ABB RAPID module: Module1.mod

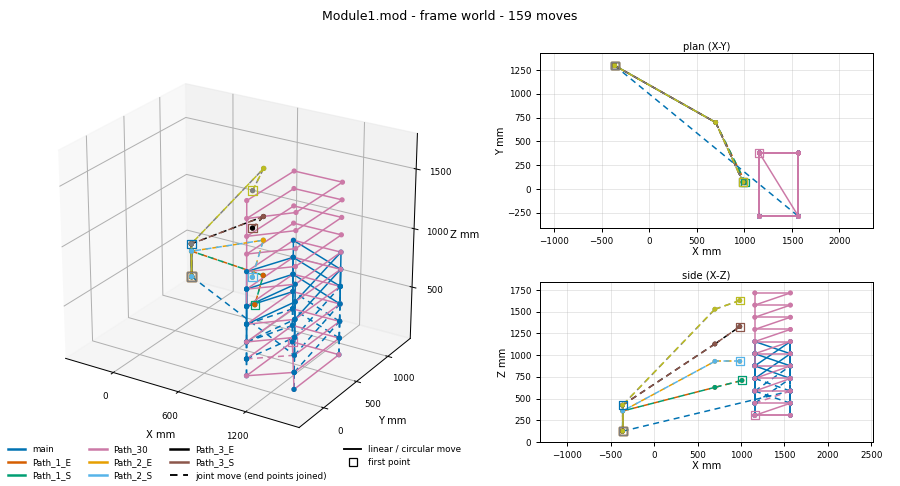
[picture p0: tool path of Module1.mod in frame world, 159 of 159 moves have a stored position in this frame; points joined in program order, loops and branches not executed]
MODULE Module1
        CONST robtarget Target_10:=[[-362.824,1298.255,124.558],[0,1,0,0],[0,0,0,0],[9E+09,9E+09,9E+09,9E+09,9E+09,9E+09]];
    CONST robtarget Target_20:=[[-361.331074857,1298.255015663,357.504486712],[0.000000006,0.937903782,0.346895511,-0.000000016],[1,0,-2,0],[9E+09,9E+09,9E+09,9E+09,9E+09,9E+09]];
    CONST robtarget Target_30:=[[699.999971128,699.99999496,629.43677315],[0.000000013,0.714564003,0.699570072,0.000000004],[0,-1,-2,0],[9E+09,9E+09,9E+09,9E+09,9E+09,9E+09]];
    CONST robtarget Target_50:=[[1570,-287,307],[0,0.707106781,0.707106781,0],[-1,0,0,0],[9E+09,9E+09,9E+09,9E+09,9E+09,9E+09]];
    CONST robtarget Target_40:=[[1012.141019914,68.859882763,709.132396194],[0.000000014,0.714564001,0.699570074,0.000000028],[0,0,-3,0],[9E+09,9E+09,9E+09,9E+09,9E+09,9E+09]];
    CONST robtarget Target_10_2:=[[-362.824,1298.255,424.558],[-0.000000012,0.998529603,-0.054209154,0.000000007],[1,0,-1,0],[9E+09,9E+09,9E+09,9E+09,9E+09,9E+09]];
    CONST robtarget Target_50_3:=[[1160,378,307],[0,0.707106781,0.707106781,0],[0,0,0,0],[9E+09,9E+09,9E+09,9E+09,9E+09,9E+09]];
    CONST robtarget Target_50_2:=[[1570,378,307],[0,0.707106781,0.707106781,0],[0,0,0,0],[9E+09,9E+09,9E+09,9E+09,9E+09,9E+09]];
    CONST robtarget Target_50_4:=[[1160,-287,307],[0,0.707106781,0.707106781,0],[-1,0,0,0],[9E+09,9E+09,9E+09,9E+09,9E+09,9E+09]];
    CONST robtarget Target_60:=[[1570,-287,447],[0,0.707106781,0.707106781,0],[0,0,0,0],[9E+09,9E+09,9E+09,9E+09,9E+09,9E+09]];
    CONST robtarget Target_60_2:=[[1570,378,447],[0,0.707106781,0.707106781,0],[0,0,1,0],[9E+09,9E+09,9E+09,9E+09,9E+09,9E+09]];
    CONST robtarget Target_60_3:=[[1160,378,447],[0,0.707106781,0.707106781,0],[0,0,1,0],[9E+09,9E+09,9E+09,9E+09,9E+09,9E+09]];
    CONST robtarget Target_60_4:=[[1160,-287,447],[0,0.707106781,0.707106781,0],[-1,0,0,0],[9E+09,9E+09,9E+09,9E+09,9E+09,9E+09]];
    CONST robtarget Target_120:=[[1570.000098335,-287.000000227,586.999987936],[-0.000000001,0.707106765,0.707106797,-0.000000001],[-1,-1,0,0],[9E+09,9E+09,9E+09,9E+09,9E+09,9E+09]];
    CONST robtarget Target_120_2:=[[1570,378,587],[0,0.707106781,0.707106781,0],[0,0,1,0],[9E+09,9E+09,9E+09,9E+09,9E+09,9E+09]];
    CONST robtarget Target_120_3:=[[1160,378,587],[0,0.707106781,0.707106781,0],[0,0,1,0],[9E+09,9E+09,9E+09,9E+09,9E+09,9E+09]];
    CONST robtarget Target_120_4:=[[1160,-287,587],[0,0.707106781,0.707106781,0],[-1,0,0,0],[9E+09,9E+09,9E+09,9E+09,9E+09,9E+09]];
    CONST robtarget Target_121:=[[1570,-287,732],[0,0.707106781,0.707106781,0],[-1,0,0,0],[9E+09,9E+09,9E+09,9E+09,9E+09,9E+09]];
    CONST robtarget Target_121_2:=[[1570,378,732],[0,0.707106781,0.707106781,0],[0,0,1,0],[9E+09,9E+09,9E+09,9E+09,9E+09,9E+09]];
    CONST robtarget Target_121_3:=[[1160,378,732],[0,0.707106781,0.707106781,0],[0,0,1,0],[9E+09,9E+09,9E+09,9E+09,9E+09,9E+09]];
    CONST robtarget Target_121_4:=[[1160,-287,732],[0,0.707106781,0.707106781,0],[-1,0,0,0],[9E+09,9E+09,9E+09,9E+09,9E+09,9E+09]];
    CONST robtarget Target_122:=[[1570,-287,877],[0,0.707106781,0.707106781,0],[-1,0,0,0],[9E+09,9E+09,9E+09,9E+09,9E+09,9E+09]];
    CONST robtarget Target_122_2:=[[1570,378,877],[0,0.707106781,0.707106781,0],[0,0,1,0],[9E+09,9E+09,9E+09,9E+09,9E+09,9E+09]];
    CONST robtarget Target_122_3:=[[1160,378,877],[0,0.707106781,0.707106781,0],[0,0,1,0],[9E+09,9E+09,9E+09,9E+09,9E+09,9E+09]];
    CONST robtarget Target_122_4:=[[1160,-287,877],[0,0.707106781,0.707106781,0],[-1,0,0,0],[9E+09,9E+09,9E+09,9E+09,9E+09,9E+09]];
    CONST robtarget Target_70_2:=[[699.999994937,700.000110159,929.436793547],[-0.000000013,0.714564003,0.699570072,0.000000004],[0,-1,-2,0],[9E+09,9E+09,9E+09,9E+09,9E+09,9E+09]];
    CONST robtarget Target_40_2:=[[987.25590411,72.978878039,929.436817205],[0.00000003,0.714563992,0.699570083,0.000000024],[0,-1,1,0],[9E+09,9E+09,9E+09,9E+09,9E+09,9E+09]];
    CONST robtarget Target_128_4:=[[1160,-287,1717],[0,0.707106781,0.707106781,0],[-1,2,-2,1],[9E+09,9E+09,9E+09,9E+09,9E+09,9E+09]];
    CONST robtarget Target_128_3:=[[1160,378,1717],[0,0.707106781,0.707106781,0],[0,0,1,0],[9E+09,9E+09,9E+09,9E+09,9E+09,9E+09]];
    CONST robtarget Target_128_2:=[[1570,378,1717],[0,0.707106781,0.707106781,0],[0,0,1,0],[9E+09,9E+09,9E+09,9E+09,9E+09,9E+09]];
    CONST robtarget Target_128:=[[1570,-287,1717],[0,0.707106781,0.707106781,0],[-1,0,0,0],[9E+09,9E+09,9E+09,9E+09,9E+09,9E+09]];
    CONST robtarget Target_127_4:=[[1160,-287,1577],[0,0.707106781,0.707106781,0],[-1,0,0,0],[9E+09,9E+09,9E+09,9E+09,9E+09,9E+09]];
    CONST robtarget Target_127_3:=[[1160,378,1577],[0,0.707106781,0.707106781,0],[0,0,1,0],[9E+09,9E+09,9E+09,9E+09,9E+09,9E+09]];
    CONST robtarget Target_127_2:=[[1570,378,1577],[0,0.707106781,0.707106781,0],[0,0,1,0],[9E+09,9E+09,9E+09,9E+09,9E+09,9E+09]];
    CONST robtarget Target_127:=[[1570,-287,1577],[0,0.707106781,0.707106781,0],[-1,0,0,0],[9E+09,9E+09,9E+09,9E+09,9E+09,9E+09]];
    CONST robtarget Target_126_4:=[[1160,-287,1437],[0,0.707106781,0.707106781,0],[-1,0,0,0],[9E+09,9E+09,9E+09,9E+09,9E+09,9E+09]];
    CONST robtarget Target_126_3:=[[1160,378,1437],[0,0.707106781,0.707106781,0],[0,0,1,0],[9E+09,9E+09,9E+09,9E+09,9E+09,9E+09]];
    CONST robtarget Target_126_2:=[[1570,378,1437],[0,0.707106781,0.707106781,0],[0,0,1,0],[9E+09,9E+09,9E+09,9E+09,9E+09,9E+09]];
    CONST robtarget Target_126:=[[1570,-287,1437],[0,0.707106781,0.707106781,0],[-1,0,0,0],[9E+09,9E+09,9E+09,9E+09,9E+09,9E+09]];
    CONST robtarget Target_125_4:=[[1160,-287,1297],[0,0.707106781,0.707106781,0],[-1,0,0,0],[9E+09,9E+09,9E+09,9E+09,9E+09,9E+09]];
    CONST robtarget Target_125_3:=[[1160,378,1297],[0,0.707106781,0.707106781,0],[0,0,1,0],[9E+09,9E+09,9E+09,9E+09,9E+09,9E+09]];
    CONST robtarget Target_125_2:=[[1570,378,1297],[0,0.707106781,0.707106781,0],[0,0,1,0],[9E+09,9E+09,9E+09,9E+09,9E+09,9E+09]];
    CONST robtarget Target_125:=[[1570,-287,1297],[0,0.707106781,0.707106781,0],[-1,0,0,0],[9E+09,9E+09,9E+09,9E+09,9E+09,9E+09]];
    CONST robtarget Target_124_4:=[[1160,-287,1157],[0,0.707106781,0.707106781,0],[-1,0,0,0],[9E+09,9E+09,9E+09,9E+09,9E+09,9E+09]];
    CONST robtarget Target_124_3:=[[1160,378,1157],[0,0.707106781,0.707106781,0],[0,0,1,0],[9E+09,9E+09,9E+09,9E+09,9E+09,9E+09]];
    CONST robtarget Target_124_2:=[[1570,378,1157],[0,0.707106781,0.707106781,0],[0,0,1,0],[9E+09,9E+09,9E+09,9E+09,9E+09,9E+09]];
    CONST robtarget Target_124:=[[1570,-287,1157],[0,0.707106781,0.707106781,0],[-1,0,0,0],[9E+09,9E+09,9E+09,9E+09,9E+09,9E+09]];
    CONST robtarget Target_123_4:=[[1160,-287,1017],[0,0.707106781,0.707106781,0],[-1,0,0,0],[9E+09,9E+09,9E+09,9E+09,9E+09,9E+09]];
    CONST robtarget Target_123_3:=[[1160,378,1017],[0,0.707106781,0.707106781,0],[0,0,1,0],[9E+09,9E+09,9E+09,9E+09,9E+09,9E+09]];
    CONST robtarget Target_123_2:=[[1570,378,1017],[0,0.707106781,0.707106781,0],[0,0,1,0],[9E+09,9E+09,9E+09,9E+09,9E+09,9E+09]];
    CONST robtarget Target_123:=[[1570,-287,1017],[0,0.707106781,0.707106781,0],[-1,0,0,0],[9E+09,9E+09,9E+09,9E+09,9E+09,9E+09]];
    CONST robtarget Target_30_2:=[[699.999992444,700.000011939,1129.436971585],[0.000000013,0.714563994,0.699570081,-0.000000007],[0,-1,-3,0],[9E+09,9E+09,9E+09,9E+09,9E+09,9E+09]];
    CONST robtarget Target_40_2_2:=[[987.255899553,72.978877702,1329.437041905],[0.00000002,0.714563994,0.699570081,0.000000013],[0,-1,1,0],[9E+09,9E+09,9E+09,9E+09,9E+09,9E+09]];
    CONST robtarget Target_10_4:=[[-362.824,1298.255,124.558],[0,1,0,0],[0,0,0,0],[9E+09,9E+09,9E+09,9E+09,9E+09,9E+09]];
    CONST robtarget Target_10_2_3:=[[-362.824,1298.255,424.558],[0,1,0,0],[1,0,-1,0],[9E+09,9E+09,9E+09,9E+09,9E+09,9E+09]];
    CONST robtarget Target_20_3:=[[123.294942114,850.000075451,439.015995707],[0.000000012,1,-0.000000212,0.000000031],[0,-1,-2,0],[9E+09,9E+09,9E+09,9E+09,9E+09,9E+09]];
    CONST robtarget Target_30_3:=[[699.999994518,700.000014013,1529.436978926],[0.000000013,0.714563998,0.699570077,0.000000012],[0,-1,-3,0],[9E+09,9E+09,9E+09,9E+09,9E+09,9E+09]];
    CONST robtarget Target_40_2_3:=[[987.255908383,72.978882952,1629.436986878],[-0.000000004,0.714563993,0.699570082,0.000000014],[0,0,1,0],[9E+09,9E+09,9E+09,9E+09,9E+09,9E+09]];
    CONST robtarget Target_20_2:=[[123.294942114,850.000075451,439.015995707],[0.000000013,0.714564003,0.699570072,0.000000004],[0,0,1,0],[9E+09,9E+09,9E+09,9E+09,9E+09,9E+09]];
    CONST robtarget Target_70:=[[700.00000486,700.000107801,929.436838226],[0.000000013,0.714563971,0.699570104,-0.000000014],[0,-1,-3,0],[9E+09,9E+09,9E+09,9E+09,9E+09,9E+09]];
!***********************************************************
    !
    ! Módulo:  Module1
    !
    ! Descripción:
    !   <Introduzca la descripción aquí>
    !
    ! Autor: deste
    !
    ! Versión: 1.0
    !
    !***********************************************************


    !***********************************************************
    !
    ! Procedimiento Main
    !
    !   Este es el punto de entrada de su programa
    !
    !***********************************************************
    PROC main()
        set Soltar;
        Reset Soltar;
        WaitDI Canasta_ok,1;
        MoveJ Target_10_2,v800,z100,Gripper\WObj:=Workobject_1;
        MoveL Target_10,v800,z100,Gripper\WObj:=Workobject_1;
        WaitUntil \InPos, Canasta_ok = 1;
        Set Agarrar;
        WaitDI Agarrado,1;
        Path_1_E;
        MoveJ Target_120,v800,z100,Gripper\WObj:=Workobject_1;
        MoveJ Target_60,v800,z10,Gripper\WObj:=Workobject_1;
        Reset Pallet;
        MoveJ Target_50,v800,z10,Gripper\WObj:=Workobject_1;
        WaitUntil \InPos, Canasta_ok = 0;
        Reset Agarrar;
        Set Soltar;
        Reset Soltar;
        MoveJ Target_60,v800,z100,Gripper\WObj:=Workobject_1;
        Path_1_S;
        !!! --------------------------- !!!
        WaitUntil \InPos, Canasta_ok = 1;
        Set Agarrar;
        WaitDI Agarrado,1;
        Path_1_E;
        MoveJ Target_120_2,v800,z100,Gripper\WObj:=Workobject_1;
        MoveJ Target_60_2,v800,z10,Gripper\WObj:=Workobject_1;
        Reset Pallet;
        MoveJ Target_50_2,v300,z10,Gripper\WObj:=Workobject_1;
        WaitUntil \InPos, Canasta_ok = 0;
        Reset Agarrar;
        Set Soltar;
        MoveJ Target_60_2,v800,z100,Gripper\WObj:=Workobject_1;
        Path_1_S;
        Reset Soltar;
        !!!-----------------------------!!!
        WaitUntil \InPos, Canasta_ok = 1;
        Set Agarrar;
        WaitDI Agarrado,1;
        Path_1_E;
        MoveJ Target_120_3,v800,z100,Gripper\WObj:=Workobject_1;
        MoveJ Target_60_3,v800,z10,Gripper\WObj:=Workobject_1;
        Reset Pallet;
        MoveJ Target_50_3,v300,z10,Gripper\WObj:=Workobject_1;
        WaitUntil \InPos, Canasta_ok = 0;
        Reset Agarrar;
        Set Soltar;
        MoveJ Target_60_3,v800,z100,Gripper\WObj:=Workobject_1;
        Path_1_S;
        Reset Soltar;
        !!!-----------------------------!!!
        WaitUntil \InPos, Canasta_ok = 1;
        Set Agarrar;
        WaitDI Agarrado,1;
        Path_1_E;
        MoveJ Target_120_4,v800,z100,Gripper\WObj:=Workobject_1;
        MoveJ Target_60_4,v800,z10,Gripper\WObj:=Workobject_1;
        Reset Pallet;
        MoveJ Target_50_4,v300,z10,Gripper\WObj:=Workobject_1;
        WaitUntil \InPos, Canasta_ok = 0;
        Reset Agarrar;
        Set Soltar;
        MoveJ Target_60_4,v800,z100,Gripper\WObj:=Workobject_1;
        Path_1_S;
        Reset Soltar;
        !!!-----------------------------!!! Segunda Bandeja
        WaitUntil \InPos, Canasta_ok = 1;
        Set Agarrar;
        WaitDI Agarrado,1;
        Path_1_E;
        MoveJ Target_121,v800,z100,Gripper\WObj:=Workobject_1;
        MoveJ Target_120,v800,z10,Gripper\WObj:=Workobject_1;
        Reset Pallet;
        MoveJ Target_60,v800,z10,Gripper\WObj:=Workobject_1;
        WaitUntil \InPos, Canasta_ok = 0;
        Reset Agarrar;
        Set Soltar;
        Reset Soltar;
        MoveJ Target_120,v800,z100,Gripper\WObj:=Workobject_1;
        Path_1_S;
        !!! --------------------------- !!!
        WaitUntil \InPos, Canasta_ok = 1;
        Set Agarrar;
        WaitDI Agarrado,1;
        Path_1_E;
        MoveJ Target_121_2,v800,z100,Gripper\WObj:=Workobject_1;
        MoveJ Target_120_2,v800,z10,Gripper\WObj:=Workobject_1;
        Reset Pallet;
        MoveJ Target_60_2,v300,z10,Gripper\WObj:=Workobject_1;
        WaitUntil \InPos, Canasta_ok = 0;
        Reset Agarrar;
        Set Soltar;
        MoveJ Target_120_2,v800,z100,Gripper\WObj:=Workobject_1;
        Path_1_S;
        Reset Soltar;
        !!!-----------------------------!!!
        WaitUntil \InPos, Canasta_ok = 1;
        Set Agarrar;
        WaitDI Agarrado,1;
        Path_1_E;
        MoveJ Target_121_3,v800,z100,Gripper\WObj:=Workobject_1;
        MoveJ Target_120_3,v800,z10,Gripper\WObj:=Workobject_1;
        Reset Pallet;
        MoveJ Target_60_3,v300,z10,Gripper\WObj:=Workobject_1;
        WaitUntil \InPos, Canasta_ok = 0;
        Reset Agarrar;
        Set Soltar;
        MoveJ Target_120_3,v800,z100,Gripper\WObj:=Workobject_1;
        Path_1_S;
        Reset Soltar;
        !!!-----------------------------!!!
        WaitUntil \InPos, Canasta_ok = 1;
        Set Agarrar;
        WaitDI Agarrado,1;
        Path_1_E;
        MoveJ Target_121_4,v800,z100,Gripper\WObj:=Workobject_1;
        MoveJ Target_120_4,v800,z10,Gripper\WObj:=Workobject_1;
        Reset Pallet;
        MoveJ Target_60_4,v300,z10,Gripper\WObj:=Workobject_1;
        WaitUntil \InPos, Canasta_ok = 0;
        Reset Agarrar;
        Set Soltar;
        MoveJ Target_120_4,v800,z100,Gripper\WObj:=Workobject_1;
        Path_1_S;
        Reset Soltar;
        !!!-----------------------------!!! Tercera Bandeja
        WaitUntil \InPos, Canasta_ok = 1;
        Set Agarrar;
        WaitDI Agarrado,1;
        Path_2_E;
        MoveJ Target_122,v800,z100,Gripper\WObj:=Workobject_1;
        MoveJ Target_121,v800,z10,Gripper\WObj:=Workobject_1;
        Reset Pallet;
        MoveL Target_120,v800,z10,Gripper\WObj:=Workobject_1;
        WaitUntil \InPos, Canasta_ok = 0;
        Reset Agarrar;
        Set Soltar;
        Reset Soltar;
        MoveJ Target_121,v800,z100,Gripper\WObj:=Workobject_1;
        Path_2_S;
        !!! --------------------------- !!!
        WaitUntil \InPos, Canasta_ok = 1;
        Set Agarrar;
        WaitDI Agarrado,1;
        Path_2_E;
        MoveJ Target_122_2,v800,z100,Gripper\WObj:=Workobject_1;
        MoveJ Target_121_2,v800,z10,Gripper\WObj:=Workobject_1;
        Reset Pallet;
        MoveJ Target_120_2,v300,z10,Gripper\WObj:=Workobject_1;
        WaitUntil \InPos, Canasta_ok = 0;
        Reset Agarrar;
        Set Soltar;
        MoveJ Target_121_2,v800,z100,Gripper\WObj:=Workobject_1;
        Path_2_S;
        Reset Soltar;
        !!!-----------------------------!!!
        WaitUntil \InPos, Canasta_ok = 1;
        Set Agarrar;
        WaitDI Agarrado,1;
        Path_2_E;
        MoveL Target_122_3,v800,z100,Gripper\WObj:=Workobject_1;
        MoveL Target_121_3,v800,z10,Gripper\WObj:=Workobject_1;
        Reset Pallet;
        MoveL Target_120_3,v300,z10,Gripper\WObj:=Workobject_1;
        WaitUntil \InPos, Canasta_ok = 0;
        Reset Agarrar;
        Set Soltar;
        MoveL Target_121_3,v800,z100,Gripper\WObj:=Workobject_1;
        Path_2_S;
        Reset Soltar;
        !!!-----------------------------!!!
        WaitUntil \InPos, Canasta_ok = 1;
        Set Agarrar;
        WaitDI Agarrado,1;
        Path_2_E;
        MoveL Target_122_4,v800,z100,Gripper\WObj:=Workobject_1;
        MoveL Target_121_4,v800,z10,Gripper\WObj:=Workobject_1;
        Reset Pallet;
        MoveL Target_120_4,v300,z10,Gripper\WObj:=Workobject_1;
        WaitUntil \InPos, Canasta_ok = 0;
        Reset Agarrar;
        Set Soltar;
        MoveL Target_121_4,v800,z100,Gripper\WObj:=Workobject_1;
        Path_2_S;
        Reset Soltar;
        !!!-----------------------------!!! Cuarta Bandeja
        WaitUntil \InPos, Canasta_ok = 1;
        Set Agarrar;
        WaitDI Agarrado,1;
        Path_2_E;
        MoveL Target_123,v800,z100,Gripper\WObj:=Workobject_1;
        MoveL Target_122,v800,z10,Gripper\WObj:=Workobject_1;
        Reset Pallet;
        MoveL Target_121,v800,z10,Gripper\WObj:=Workobject_1;
        WaitUntil \InPos, Canasta_ok = 0;
        Reset Agarrar;
        Set Soltar;
        Reset Soltar;
        MoveL Target_122,v800,z100,Gripper\WObj:=Workobject_1;
        Path_2_S;
        !!! --------------------------- !!!
        WaitUntil \InPos, Canasta_ok = 1;
        Set Agarrar;
        WaitDI Agarrado,1;
        Path_2_E;
        MoveL Target_123_2,v800,z100,Gripper\WObj:=Workobject_1;
        MoveL Target_122_2,v800,z10,Gripper\WObj:=Workobject_1;
        Reset Pallet;
        MoveL Target_121_2,v300,z10,Gripper\WObj:=Workobject_1;
        WaitUntil \InPos, Canasta_ok = 0;
        Reset Agarrar;
        Set Soltar;
        MoveL Target_122_2,v800,z100,Gripper\WObj:=Workobject_1;
        Path_2_S;
        Reset Soltar;
        !!!-----------------------------!!!
        WaitUntil \InPos, Canasta_ok = 1;
        Set Agarrar;
        WaitDI Agarrado,1;
        Path_2_E;
        MoveL Target_123_3,v800,z100,Gripper\WObj:=Workobject_1;
        MoveL Target_122_3,v800,z10,Gripper\WObj:=Workobject_1;
        Reset Pallet;
        MoveL Target_121_3,v300,z10,Gripper\WObj:=Workobject_1;
        WaitUntil \InPos, Canasta_ok = 0;
        Reset Agarrar;
        Set Soltar;
        MoveL Target_122_3,v800,z100,Gripper\WObj:=Workobject_1;
        Path_2_S;
        Reset Soltar;
        !!!-----------------------------!!!
        WaitUntil \InPos, Canasta_ok = 1;
        Set Agarrar;
        WaitDI Agarrado,1;
        Path_2_E;
        MoveL Target_123_4,v800,z100,Gripper\WObj:=Workobject_1;
        MoveL Target_122_4,v800,z10,Gripper\WObj:=Workobject_1;
        Reset Pallet;
        MoveL Target_121_4,v300,z10,Gripper\WObj:=Workobject_1;
        WaitUntil \InPos, Canasta_ok = 0;
        Reset Agarrar;
        Set Soltar;
        MoveL Target_122_4,v800,z100,Gripper\WObj:=Workobject_1;
        Path_2_S;
        Reset Soltar;
        !!!-----------------------------!!! Quinta Bandeja
        WaitUntil \InPos, Canasta_ok = 1;
        Set Agarrar;
        WaitDI Agarrado,1;
        Path_3_E;
        MoveL Target_124,v800,z100,Gripper\WObj:=Workobject_1;
        MoveL Target_123,v800,z10,Gripper\WObj:=Workobject_1;
        Reset Pallet;
        MoveL Target_122,v800,z10,Gripper\WObj:=Workobject_1;
        WaitUntil \InPos, Canasta_ok = 0;
        Reset Agarrar;
        Set Soltar;
        Reset Soltar;
        MoveL Target_123,v800,z100,Gripper\WObj:=Workobject_1;
        Path_3_S;
        !!! --------------------------- !!!
        WaitUntil \InPos, Canasta_ok = 1;
        Set Agarrar;
        WaitDI Agarrado,1;
        Path_3_E;
        MoveL Target_124_2,v800,z100,Gripper\WObj:=Workobject_1;
        MoveL Target_123_2,v800,z10,Gripper\WObj:=Workobject_1;
        Reset Pallet;
        MoveL Target_122_2,v300,z10,Gripper\WObj:=Workobject_1;
        WaitUntil \InPos, Canasta_ok = 0;
        Reset Agarrar;
        Set Soltar;
        MoveL Target_123_2,v800,z100,Gripper\WObj:=Workobject_1;
        Path_3_S;
        Reset Soltar;
        !!!-----------------------------!!!
        WaitUntil \InPos, Canasta_ok = 1;
        Set Agarrar;
        WaitDI Agarrado,1;
        Path_3_E;
        MoveL Target_124_3,v800,z100,Gripper\WObj:=Workobject_1;
        MoveL Target_123_3,v800,z10,Gripper\WObj:=Workobject_1;
        Reset Pallet;
        MoveL Target_122_3,v300,z10,Gripper\WObj:=Workobject_1;
        WaitUntil \InPos, Canasta_ok = 0;
        Reset Agarrar;
        Set Soltar;
        MoveL Target_123_3,v800,z100,Gripper\WObj:=Workobject_1;
        Path_3_S;
        Reset Soltar;
        !!!-----------------------------!!!
        WaitUntil \InPos, Canasta_ok = 1;
        Set Agarrar;
        WaitDI Agarrado,1;
        Path_3_E;
        MoveL Target_124_4,v800,z100,Gripper\WObj:=Workobject_1;
        MoveL Target_123_4,v800,z10,Gripper\WObj:=Workobject_1;
        Reset Pallet;
        MoveL Target_122_4,v300,z10,Gripper\WObj:=Workobject_1;
        WaitUntil \InPos, Canasta_ok = 0;
        Reset Agarrar;
        Set Soltar;
        MoveL Target_123_4,v800,z100,Gripper\WObj:=Workobject_1;
        Path_3_S;
        Reset Soltar;
    ENDPROC

    PROC Path_1_E()
        MoveL Target_10,v1000,z100,Gripper\WObj:=Workobject_1;
        MoveJ Target_20,v1000,z100,Gripper\WObj:=Workobject_1;
        MoveJ Target_30,v1000,z100,Gripper\WObj:=Workobject_1;
        MoveJ Target_40,v1000,z100,Gripper\WObj:=Workobject_1;
    ENDPROC
    PROC Path_1_S()
        MoveJ Target_40,v1000,z100,Gripper\WObj:=Workobject_1;
        MoveJ Target_30,v800,z100,Gripper\WObj:=Workobject_1;
        MoveJ Target_20,v1000,z100,Gripper\WObj:=Workobject_1;
        MoveJ Target_10,v600,z100,Gripper\WObj:=Workobject_1;
    ENDPROC
    PROC Path_30()
        MoveL Target_50_3,v1000,z100,Gripper\WObj:=Workobject_1;
        MoveL Target_50,v1000,z100,Gripper\WObj:=Workobject_1;
        MoveL Target_50_2,v1000,z100,Gripper\WObj:=Workobject_1;
        MoveL Target_50_3,v1000,z100,Gripper\WObj:=Workobject_1;
        MoveL Target_50_4,v1000,z100,Gripper\WObj:=Workobject_1;
        MoveL Target_60,v1000,z100,Gripper\WObj:=Workobject_1;
        MoveL Target_60_2,v1000,z100,Gripper\WObj:=Workobject_1;
        MoveL Target_60_3,v1000,z100,Gripper\WObj:=Workobject_1;
        MoveL Target_60_4,v1000,z100,Gripper\WObj:=Workobject_1;
        MoveJ Target_120,v1000,z100,Gripper\WObj:=Workobject_1;
        MoveL Target_120_2,v1000,z100,Gripper\WObj:=Workobject_1;
        MoveL Target_120_3,v1000,z100,Gripper\WObj:=Workobject_1;
        MoveL Target_120_4,v1000,z100,Gripper\WObj:=Workobject_1;
        MoveL Target_121,v1000,z100,Gripper\WObj:=Workobject_1;
        MoveL Target_121_2,v1000,z100,Gripper\WObj:=Workobject_1;
        MoveL Target_121_3,v1000,z100,Gripper\WObj:=Workobject_1;
        MoveL Target_121_4,v1000,z100,Gripper\WObj:=Workobject_1;
        MoveL Target_122,v1000,z100,Gripper\WObj:=Workobject_1;
        MoveL Target_122_2,v1000,z100,Gripper\WObj:=Workobject_1;
        MoveL Target_122_3,v1000,z100,Gripper\WObj:=Workobject_1;
        MoveL Target_122_4,v1000,z100,Gripper\WObj:=Workobject_1;
        MoveL Target_128_4,v1000,z100,Gripper\WObj:=Workobject_1;
        MoveL Target_128_3,v1000,z100,Gripper\WObj:=Workobject_1;
        MoveL Target_128_2,v1000,z100,Gripper\WObj:=Workobject_1;
        MoveL Target_128,v1000,z100,Gripper\WObj:=Workobject_1;
        MoveL Target_127_4,v1000,z100,Gripper\WObj:=Workobject_1;
        MoveL Target_127_3,v1000,z100,Gripper\WObj:=Workobject_1;
        MoveL Target_127_2,v1000,z100,Gripper\WObj:=Workobject_1;
        MoveL Target_127,v1000,z100,Gripper\WObj:=Workobject_1;
        MoveL Target_126_4,v1000,z100,Gripper\WObj:=Workobject_1;
        MoveL Target_126_3,v1000,z100,Gripper\WObj:=Workobject_1;
        MoveL Target_126_2,v1000,z100,Gripper\WObj:=Workobject_1;
        MoveL Target_126,v1000,z100,Gripper\WObj:=Workobject_1;
        MoveL Target_125_4,v1000,z100,Gripper\WObj:=Workobject_1;
        MoveL Target_125_3,v1000,z100,Gripper\WObj:=Workobject_1;
        MoveL Target_125_2,v1000,z100,Gripper\WObj:=Workobject_1;
        MoveL Target_125,v1000,z100,Gripper\WObj:=Workobject_1;
        MoveL Target_124_4,v1000,z100,Gripper\WObj:=Workobject_1;
        MoveL Target_124_3,v1000,z100,Gripper\WObj:=Workobject_1;
        MoveL Target_124_2,v1000,z100,Gripper\WObj:=Workobject_1;
        MoveL Target_124,v1000,z100,Gripper\WObj:=Workobject_1;
        MoveL Target_123_4,v1000,z100,Gripper\WObj:=Workobject_1;
        MoveL Target_123_3,v1000,z100,Gripper\WObj:=Workobject_1;
        MoveL Target_123_2,v1000,z100,Gripper\WObj:=Workobject_1;
        MoveL Target_123,v1000,z100,Gripper\WObj:=Workobject_1;
    ENDPROC
    PROC Path_2_E()
        MoveL Target_10,v1000,z100,Gripper\WObj:=Workobject_1;
        MoveJ Target_20,v1000,z100,Gripper\WObj:=Workobject_1;
        MoveJ Target_70,v1000,z100,Gripper\WObj:=Workobject_1;
        MoveJ Target_40_2,v1000,z100,Gripper\WObj:=Workobject_1;
    ENDPROC
    PROC Path_2_S()
        MoveL Target_40_2,v1000,z100,Gripper\WObj:=Workobject_1;
        MoveJ Target_70,v1000,z100,Gripper\WObj:=Workobject_1;
        MoveJ Target_20,v1000,z100,Gripper\WObj:=Workobject_1;
        MoveJ Target_10,v1000,z100,Gripper\WObj:=Workobject_1;
    ENDPROC
    PROC Path_3_E()
        MoveL Target_10,v1000,z100,Gripper\WObj:=Workobject_1;
        MoveL Target_10_2,v1000,z100,Gripper\WObj:=Workobject_1;
        MoveJ Target_30_2,v1000,z100,Gripper\WObj:=Workobject_1;
        MoveJ Target_40_2_2,v1000,z100,Gripper\WObj:=Workobject_1;
    ENDPROC
    PROC Path_3_S()
        MoveL Target_40_2_2,v1000,z100,Gripper\WObj:=Workobject_1;
        MoveJ Target_30_2,v1000,z100,Gripper\WObj:=Workobject_1;
        MoveJ Target_10_2,v1000,z100,Gripper\WObj:=Workobject_1;
        MoveL Target_10,v1000,z100,Gripper\WObj:=Workobject_1;
    ENDPROC
    PROC Path_4_E()
        MoveL Target_10_4,v1000,z100,Gripper\WObj:=Workobject_1;
        MoveL Target_10_2,v1000,z100,Gripper\WObj:=Workobject_1;
        MoveJ Target_30_3,v1000,z100,Gripper\WObj:=Workobject_1;
        MoveJ Target_40_2_3,v1000,z100,Gripper\WObj:=Workobject_1;
    ENDPROC
    PROC Path_4_S()
        MoveL Target_40_2_3,v1000,z100,Gripper\WObj:=Workobject_1;
        MoveJ Target_30_3,v1000,z100,Gripper\WObj:=Workobject_1;
        MoveJ Target_10_2,v1000,z100,Gripper\WObj:=Workobject_1;
        MoveL Target_10_4,v1000,z100,Gripper\WObj:=Workobject_1;
    ENDPROC


ENDMODULE
